FUNCTION_BLOCK CruiseController_FBDKInterface (* Basic Function Block Type *)
  (* Standard: 61499-2 *)
  (* Version 0.2, 2003-12-04, JHC, Rockwell Automation, Renamed for better indexing. *)
  (* Version 0.1, 2002-11-05, JHC, Rockwell Automation, Corrected missing ST element in Algorithm REQ. *)
  (* Version 0.0, 2000-05-30, JHC, Rockwell Automation *)
  (* Compiler header: package fb.rt.benchmarks.cruisecontrol; *)
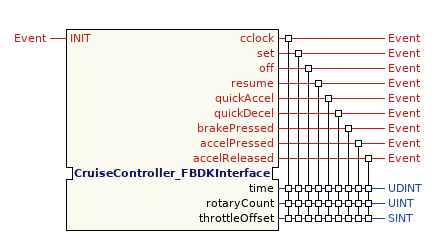
  EVENT_INPUT
    INIT; (* Initialization Request *)
  END_EVENT
  EVENT_OUTPUT
    cclock WITH time, rotaryCount, throttleOffset;
    set WITH time, rotaryCount, throttleOffset;
    off WITH time, rotaryCount, throttleOffset;
    resume WITH time, rotaryCount, throttleOffset;
    quickAccel WITH time, rotaryCount, throttleOffset;
    quickDecel WITH time, rotaryCount, throttleOffset;
    brakePressed WITH time, rotaryCount, throttleOffset;
    accelPressed WITH time, rotaryCount, throttleOffset;
    accelReleased WITH time, rotaryCount, throttleOffset;
  END_EVENT
  VAR_OUTPUT
    time : UDINT; (* 10ms tick *)
    rotaryCount : UINT;
    throttleOffset : SINT;
  END_VAR
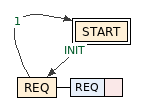
  EC_STATES
    START; (* Initial State *)
    REQ : REQ; (* Normal execution *)
  END_STATES
  EC_TRANSITIONS
    START TO REQ := INIT;
    REQ TO START := 1;
  END_TRANSITIONS
  ALGORITHM REQ IN Java: (* Normally executed algorithm *)
// Fire randomly generated inputs into the system
final File file = new File("src" + File.separator + "benchmarks" + File.separator + "Vectors" + File.separator +"CruiseController_Vector.txt");
BufferedReader testVector = null;
Integer tempInt = new Integer(0);
String inputPath = file.getAbsolutePath();
System.out.println();
System.out.println("Full Test using: " + inputPath);
int testLoop = 0;
long totalTime = 0;
long avgFull = 0;
boolean TestBenchOnly = false;
for(testLoop = 0; testLoop < 30; testLoop++)
{
if( testLoop == 15 )
{
// End of full testing
TestBenchOnly = true;
avgFull = (totalTime / 15);
System.out.println("\nAverage = " + avgFull);
totalTime = 0;
System.out.println("\n\nTestBench Only using: " + inputPath);

}


try
{
testVector = new BufferedReader(new FileReader(inputPath));
}
catch (FileNotFoundException e)
{
e.printStackTrace();
}
// RUN TEST
try
{
String line;
long startTime = System.nanoTime();
while ((line = testVector.readLine()) != null)
{
 String inputs[] = line.split(" ");

// Data first
time.value = Integer.parseInt(inputs[9]);
rotaryCount.value = Integer.parseInt(inputs[10]);
throttleOffset.value = (byte)Integer.parseInt(inputs[11]);


if( inputs[0].equals("1"))
{
if( !TestBenchOnly )
cclock.serviceEvent(this);
}
if( inputs[1].equals("1"))
{
if( !TestBenchOnly )
set.serviceEvent(this);
}
if( inputs[2].equals("1"))
{
if( !TestBenchOnly )
off.serviceEvent(this);
}
if( inputs[3].equals("1"))
{
if( !TestBenchOnly )
resume.serviceEvent(this);
}
if( inputs[4].equals("1"))
{
if( !TestBenchOnly )
quickAccel.serviceEvent(this);
}
if( inputs[5].equals("1"))
{
if( !TestBenchOnly )
quickDecel.serviceEvent(this);
}
if( inputs[6].equals("1"))
{
if( !TestBenchOnly )
brakePressed.serviceEvent(this);
}
if( inputs[7].equals("1"))
{
if( !TestBenchOnly )
accelPressed.serviceEvent(this);
}
if( inputs[8].equals("1"))
{
if( !TestBenchOnly )
accelReleased.serviceEvent(this);
}


}
long endTime = System.nanoTime();
System.out.printf("Time taken: %d\n", endTime - startTime);
totalTime += endTime - startTime;
testVector.close();
}
catch (IOException e)
{
e.printStackTrace();
}



}

// End of TestBench testing
System.out.println("\nAverage = " + (totalTime / 15));

System.out.println("\nFinal Time = " + (avgFull - (totalTime / 15)));
  END_ALGORITHM
END_FUNCTION_BLOCK
